{attribute 'qualified_only'}
{attribute 'strict'}
{attribute 'to_string'}
TYPE E_STATION_GEAR_DISTANCE_AXIS :
(
  // which axis nSync distance is checked for termination of GearInPosCA.
  // after nSync distance the station does a regular outfeed to target station
	FOLLOW_THE_MASTER,
  FOLLOW_THE_SLAVE
)UINT;
END_TYPE

(* stored: Version 1.1.0.1, ProductVersion 3.1.4026.18
   DUT E_STATION_GEAR_DISTANCE_AXIS: Id {18922e15-eb74-4aeb-a879-d437c58ec711} *)
